{attribute 'qualified_only'}
{attribute 'strict'}
{attribute 'to_string'}
TYPE E_SafeLogicState :
(
	OFFLINE 		:= 0,
	RUN				:= 1,
	STOP			:= 2,
	SAFE			:= 3,
	ERROR           := 4,
	START           := 6,
	PREPARE         := 8,
	RESTORE         := 10,
	PROJECT_CRC_OK  := 11
);
END_TYPE

(* stored: Version 1.1.0.1, ProductVersion 3.1.4024.12
   EnumerationTextList E_SafeLogicState: Id {2f1df3f9-9389-4821-bd6f-0e78743acdd8} *)
